// TIA Portal V17 export
// export: Created 2022-07-28T18:02:45.6616783Z, ExportSetting None, DisplayName Totally Integrated Automation Portal, DisplayVersion V17, DisplayName TIA Portal Openness, DisplayVersion V17, DisplayName TIA Portal Teamcenter Gateway, DisplayVersion V17, DisplayName TIA Portal Version Control Interface, DisplayVersion V17, DisplayName TIA Portal Test Suite Advanced, DisplayVersion V17, DisplayName SINAMICS Startdrive Advanced, DisplayVersion V17, DisplayName SINAMICS DCC, DisplayVersion V17, DisplayName SINAMICS Startdrive G130, G150, S120, S150, SINAMICS MV, S210, DisplayVersion V17, DisplayName SINAMICS Startdrive G110M, G120, G120C, G120D, G120P, G115D, DisplayVersion V17, DisplayName STEP 7 Professional, DisplayVersion V17, DisplayName SIMATIC Energy Suite, DisplayVersion V17, DisplayName STEP 7 CFC, DisplayVersion V17, DisplayName STEP 7 Safety, DisplayVersion V17, DisplayName WinCC Advanced / Unified PC, DisplayVersion V17, DisplayName SIMATIC Visualization Architect, DisplayVersion V17
FUNCTION_BLOCK "Lib_FB_PT1_Ramp"   // FB3, SCL
TITLE = Simulation of PT1
{ S7_Optimized_Access := 'TRUE' }
AUTHOR : VS
FAMILY : Simulation
VERSION : 2.0
// Block for simulation systems which can represetation like PT1;
//                   K
// W(p) = ----------------
//               Tp  +  1
// stored: AutoNumber false, MemoryReserve 100, SetENOAutomatically false
   VAR_INPUT
      i_Reset : Bool;   // 1 = reset all parameters; output = input
      i_Invert : Bool;   // 1 = invert logic (cooling)
      ir_Input : Real;   // Input value
      ir_T1_sec : Real := 2.1;   // Time T1, sec
      ir_K : Real := 1.0;   // Gain K
      ir_T_cycle_sec : Real := 0.1;   // Cyclic time, s (OB time)
      ir_OffSet_Out : Real := 0.0;   // Offset for out value
      ir_Delta : Real := 0.1;
   END_VAR
   VAR_OUTPUT
      q_DataErr : Bool;   // 1 = invalid data
      qr_Output : Real;   // Output value
   END_VAR
   VAR
      s_FirstCall : Bool;   // For internal use
      sr_Output : Real;   // Output value
      sr_T1_sec_Old : Real := 1.0;   // Old value of time T1, sec
      sr_K_Old : Real := 1.0;   // Old value of Gain K
      sr_T_cycle_sec_Old : Real := 0.1;   // Old value of cyclic time, s (OB time)
      sr_InPart : Real;   // For internal use
      sr_ExpPart : Real;   // For internal use
   END_VAR
   VAR_TEMP
      tr_LogKp : Real;   // Input value for logic
   END_VAR
BEGIN
       (*
       Transfer function:
                 k
       W(p) = --------
               Tp + 1

       Equition after invers Z-transformation:

       Y[t] = Y[t-1] * e(-Tc/T1) + X[t]*K*(1-e(-Tc/T1))   

       *)

       //Invert logic checking
       IF #i_Invert
       THEN
           #tr_LogKp := -1.0 * #ir_K;
       ELSE
           #tr_LogKp := #ir_K;
       END_IF;

       //Check parameters
       IF #ir_T1_sec <= 0.0
           OR #ir_T_cycle_sec <= 0.0
       THEN
           #q_DataErr := TRUE;
           #sr_Output := 0;
           #qr_Output := 0;
           RETURN;
       ELSE
           #q_DataErr := FALSE;
       END_IF;

       //It is parts of z-equition calculation
       //We calculate only on changes or at begin
       IF NOT #s_FirstCall
           OR (#sr_T1_sec_Old <> #ir_T1_sec)
           OR (#sr_K_Old <> #tr_LogKp)
           OR (#sr_T_cycle_sec_Old <> #ir_T_cycle_sec)
       THEN
           #s_FirstCall := 1;

           //Calculation the parts of invert z-transform equition
           #sr_ExpPart := - EXP(- #ir_T_cycle_sec / #ir_T1_sec);
           #sr_InPart := #tr_LogKp * (1 + #sr_ExpPart);

           //It rewrites old values
           #sr_T1_sec_Old := #ir_T1_sec;
           #sr_K_Old := #tr_LogKp;
           #sr_T_cycle_sec_Old := #ir_T_cycle_sec;
       END_IF;

       // Differencial Equation of PT1-System for calculate output value
       #sr_Output := (#ir_Input)* #sr_InPart - #sr_Output * #sr_ExpPart;

       //if sub In-Out < delta -> Out = In
       IF ABS(#ir_Input - #sr_Output) <= #ir_Delta
       THEN
           #sr_Output := #ir_Input;
       END_IF;

       //If reset occured
       IF #i_Reset
       THEN
           #sr_Output := #ir_Input * #tr_LogKp;
       END_IF;

       //New value writes to output
       #qr_Output := #sr_Output + #ir_OffSet_Out;
END_FUNCTION_BLOCK
